PROGRAM MAIN
VAR
	in_speedstep: INT:= 1;
	in_speed: INT:= 5;
	in_maxcount: INT:= 100;
	in_increment: INT:= 1;	
	incerement: INT:= 1;
	b_IncrementNow: BOOL;
	//-----------------------------------
	b_Controll: BOOL:= FALSE;
	b_ModeSelect: BOOL:= FALSE;
	b_ConfirmNotifi: BOOL:= FALSE;
	b_LightGrid: BOOL:= TRUE;
	b_EmSwitch: BOOL:= TRUE;
	b_ScrewDoor: BOOL:= TRUE;
	i_OverAllSpeed: REAL:= 76.86;
	//----------------------------------
	i_DepragStatus: INT:= 1;
	i_DepragStep: INT:= 2;
	r_DepragTorque: REAL:= 0.86;
	i_DepragAngle: INT:= 56;
	i_DepragProgramNR: INT:= 28;
	r_DepragCycleTime: REAL:= 1.3;
	i_ErrorMessage: INT:= 0;
	//-----------------------------------
	t_temp: INT:= 0;
END_VAR

IF HMI_Variable.b_ConfirmNotifi  THEN
	HMI_Variable.b_ClearNotifi := TRUE;
	HMI_Variable.i_ErrorMessage:= 0;
END_IF

END_PROGRAM

(* stored: Version 1.1.0.1, ProductVersion 3.1.4022.7
   POU MAIN: Id {1515f92f-5de5-44c8-8eb7-b2c6bf787c06}, SpecialFunc None *)
